(* Logix 5000 project; controller cal1632 1756-L62 rev 16.20; software revision 16.05; part 17 of 57 *)
(* tags used below, declared in another part *)
   AFI : BOOL;
   FAULT : BOOL;
   p01_param_fan_zero_speed : REAL;
   p01_param_open_oven_exh_sp : REAL;
   p01_param_open_oven_temp : REAL;
   p01_recipe_active : recipe;
   p01r02 : routine;
   p01r09_open_oven : BOOL;
   p01r09_pb_global_reset : BOOL;
   p01r13_permissive_oxidizer : BOOL;
   p02_dint_from_hmi : hmi_dint;
   p11r02_shutdown_temp : BOOL;
   p11r30 : routine;
   p11r30_request_heat : BOOL;
   p12_ai_exhaust_rpm : REAL;
   p12_ai_lfl : REAL;
   p12_ai_tc01 : REAL;
   p12_ai_tc02 : REAL;
   p12_ao_cv : REAL;
   p12_ao_exhaust_selected_speed : REAL;
   p12_di_burner_auto : BOOL;
   p12_di_burner_safeties_ok : BOOL;
   p12_di_door_open : BOOL;
   p12_di_exh : acs800_di_normal;
   p12_di_exh_fan_mtr_ts : BOOL;
   p12_di_exh_flow_ok : BOOL;
   p12_di_flame_failure : BOOL;
   p12_di_flame_on : BOOL;
   p12_di_fresh_air_clean : BOOL;
   p12_di_high_limit_temp_ok : BOOL;
   p12_di_recirc : acs800_di_normal;
   p12_di_recirc_flow_ok : BOOL;
   p12_di_sp0 : BOOL;
   p12_di_sp1 : BOOL;
   p12_di_tc01_bo : BOOL;
   p12_di_tc02_bo : BOOL;
   p12_di_zone_air_clean : BOOL;
   p12_do_enable_burner : BOOL;
   p12_do_exh : acs800_do_normal;
   p12_do_rst_flame : BOOL;
   p12_param_fast_to_soak : REAL;
   p12_param_lfl_hhl : REAL;
   p12_param_lfl_hl : REAL;
   p12_param_pid1_ff : REAL;
   p12_param_pid1_kd : REAL;
   p12_param_pid1_ki : REAL;
   p12_param_pid1_kp : REAL;
   p12_param_pid2_ff : REAL;
   p12_param_pid2_kd : REAL;
   p12_param_pid2_ki : REAL;
   p12_param_pid2_kp : REAL;
   p12_param_soak_to_fast : REAL;
   p12_param_tc01_dev : REAL;
   p12_param_tc01_hl : REAL;
   p12r02_shutdown_temp : BOOL;
   p12r16_pid_temp_cv : DINT;
   p12r16_temp_ok : BOOL;
   p12r20_safeties_ok : BOOL;
   p12r20_state : DINT;
   p12r30 : routine;
   p12r30_cv_man_sp : REAL;
   p12r30_pb_auto : BOOL;
   p12r30_pb_manual : BOOL;
   p12r30_pb_zone_off : BOOL;
   p12r30_pb_zone_on : BOOL;
   p12r30_permissive_run : BOOL;
   p12r30_pid_temp : PID;
   p12r30_pid_temp_pv : REAL;
   p12r30_pid_temp_sp : REAL;
   p12r30_pid_temp_sp_error : REAL;
   p12r30_pid_temp_sp_last : REAL;
   p12r30_request_deviation_warning : BOOL;
   p12r30_request_heat : BOOL;
   p12r30_request_heat_last : BOOL;
   p12r30_request_manual : BOOL;
   p12r30_request_PID_shot : BOOL;
   p12r30_request_soak_control : BOOL;
   p12r30_temp_deviation_setpoint : DINT;
   p12r30_timer_fault : TIMER[16];
   p12r30_timer_warning : TIMER[12];
   p12r30_vfds_ok : BOOL;
   p12r31 : routine;
   p12r31_pb_start : BOOL;
   p12r31_pb_stop : BOOL;
   p12r31_request_auto_run : BOOL;
   p12r31_run_permissive : BOOL;
   p12r31_timer_fault : TIMER[5];
   p12r31_timer_warning : TIMER[5];
   p12r31_vfd_stopped : BOOL;
   p12r32 : routine;
   p23_di_exhaust_speed_ok : BOOL;
   p23_di_impreg_exhaust_running : BOOL;
   p23_di_impreg_tank_up : BOOL;
   p23_di_supply_speed_ok : BOOL;
   p23r02 : routine;
   p23r13 : routine;
(* P12_Zone_2, continued *)

ROUTINE R30_Temperature_Control   (* ladder *)
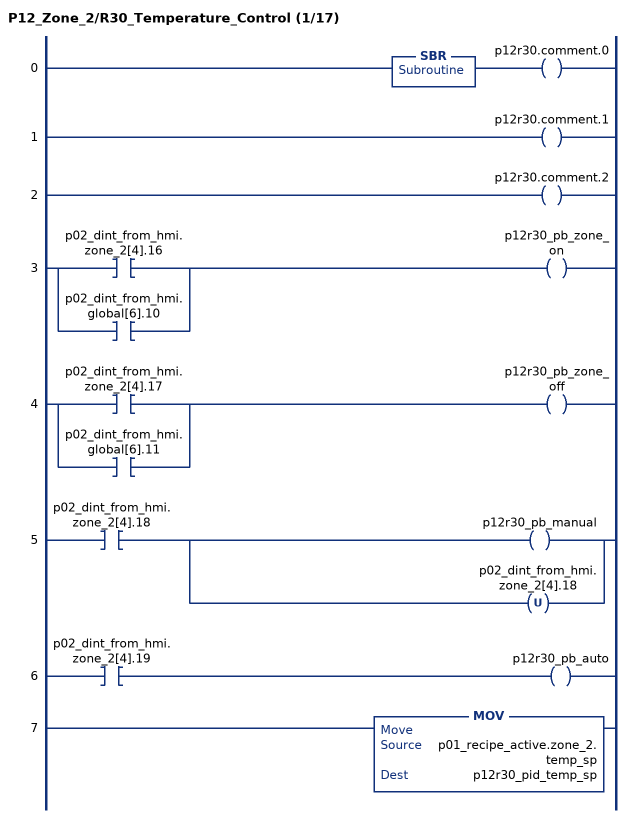
   0: SBR()OTE(p12r30.comment.0);
   1: OTE(p12r30.comment.1);
   2: OTE(p12r30.comment.2);
   3: [XIC(p02_dint_from_hmi.zone_2[4].16) ,XIC(p02_dint_from_hmi.global[6].10) ]OTE(p12r30_pb_zone_on);
   4: [XIC(p02_dint_from_hmi.zone_2[4].17) ,XIC(p02_dint_from_hmi.global[6].11) ]OTE(p12r30_pb_zone_off);
   5: XIC(p02_dint_from_hmi.zone_2[4].18)[OTE(p12r30_pb_manual) ,OTU(p02_dint_from_hmi.zone_2[4].18) ];
   6: XIC(p02_dint_from_hmi.zone_2[4].19)OTE(p12r30_pb_auto);
   7: MOV(p01_recipe_active.zone_2.temp_sp,p12r30_pid_temp_sp);
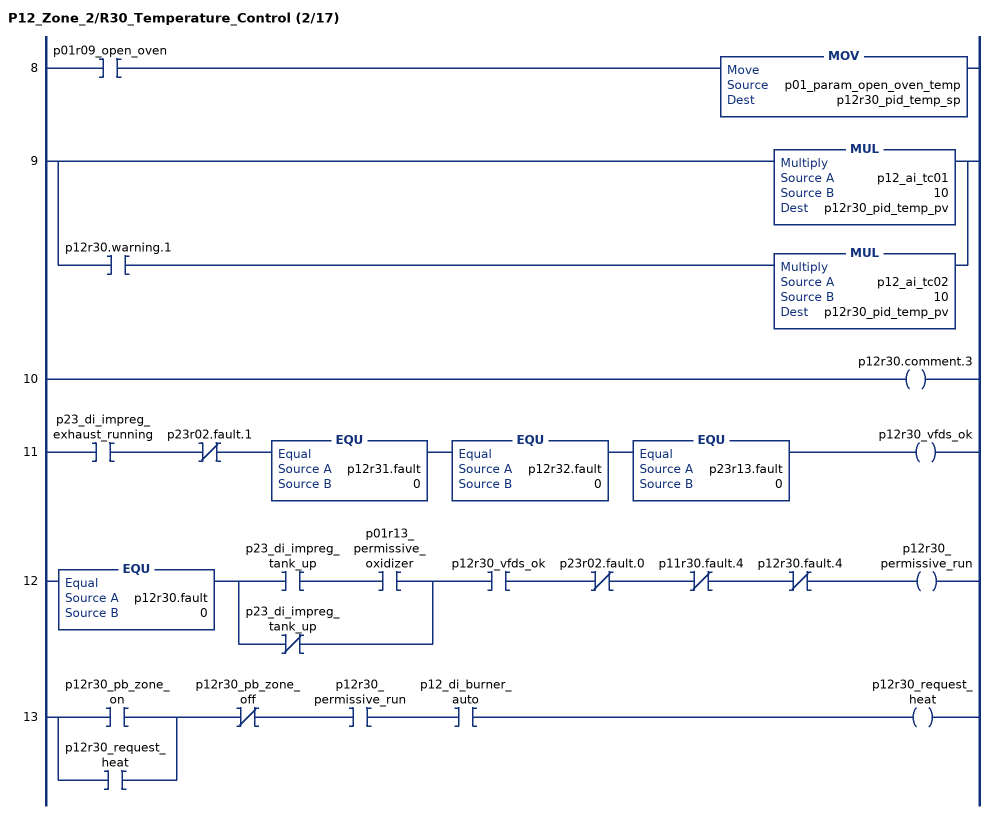
   8: XIC(p01r09_open_oven)MOV(p01_param_open_oven_temp,p12r30_pid_temp_sp);
   9: [MUL(p12_ai_tc01,10,p12r30_pid_temp_pv) ,XIC(p12r30.warning.1) MUL(p12_ai_tc02,10,p12r30_pid_temp_pv) ];
   10: OTE(p12r30.comment.3);
   11: XIC(p23_di_impreg_exhaust_running)XIO(p23r02.fault.1)EQU(p12r31.fault,0)EQU(p12r32.fault,0)EQU(p23r13.fault,0)OTE(p12r30_vfds_ok);
   12: EQU(p12r30.fault,0)[XIC(p23_di_impreg_tank_up) XIC(p01r13_permissive_oxidizer) ,XIO(p23_di_impreg_tank_up) ]XIC(p12r30_vfds_ok)XIO(p23r02.fault.0)XIO(p11r30.fault.4)XIO(p12r30.fault.4)OTE(p12r30_permissive_run);
   13: [XIC(p12r30_pb_zone_on) ,XIC(p12r30_request_heat) ]XIO(p12r30_pb_zone_off)XIC(p12r30_permissive_run)XIC(p12_di_burner_auto)OTE(p12r30_request_heat);
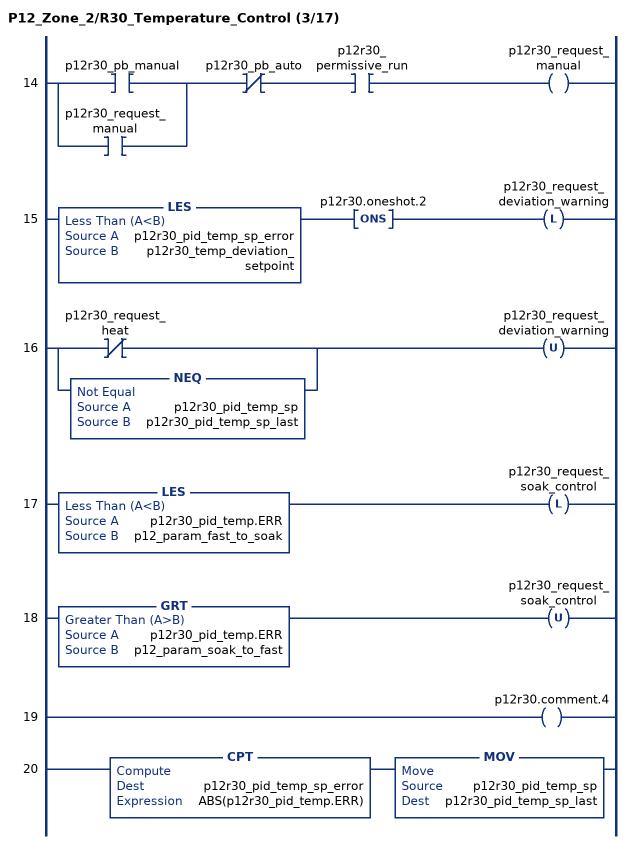
   14: [XIC(p12r30_pb_manual) ,XIC(p12r30_request_manual) ]XIO(p12r30_pb_auto)XIC(p12r30_permissive_run)OTE(p12r30_request_manual);
   15: LES(p12r30_pid_temp_sp_error,p12r30_temp_deviation_setpoint)ONS(p12r30.oneshot.2)OTL(p12r30_request_deviation_warning);
   16: [XIO(p12r30_request_heat) ,NEQ(p12r30_pid_temp_sp,p12r30_pid_temp_sp_last) ]OTU(p12r30_request_deviation_warning);
   17: LES(p12r30_pid_temp.ERR,p12_param_fast_to_soak)OTL(p12r30_request_soak_control);
   18: GRT(p12r30_pid_temp.ERR,p12_param_soak_to_fast)OTU(p12r30_request_soak_control);
   19: OTE(p12r30.comment.4);
   20: CPT(p12r30_pid_temp_sp_error,ABS(p12r30_pid_temp.ERR))MOV(p12r30_pid_temp_sp,p12r30_pid_temp_sp_last);
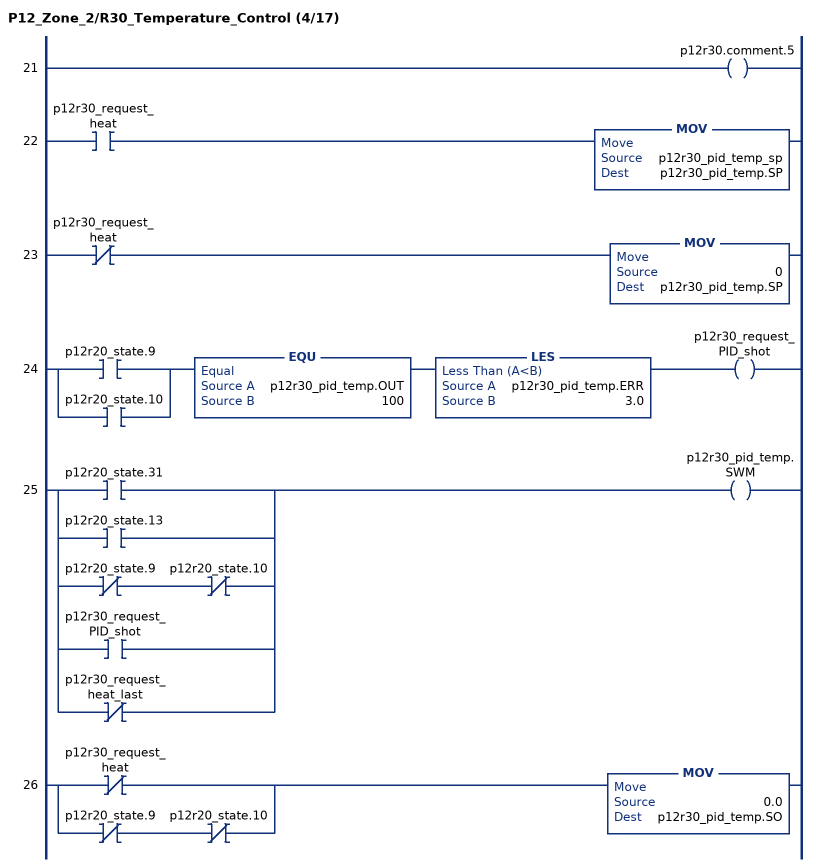
   21: OTE(p12r30.comment.5);
   22: XIC(p12r30_request_heat)MOV(p12r30_pid_temp_sp,p12r30_pid_temp.SP);
   23: XIO(p12r30_request_heat)MOV(0,p12r30_pid_temp.SP);
   24: [XIC(p12r20_state.9) ,XIC(p12r20_state.10) ]EQU(p12r30_pid_temp.OUT,100)LES(p12r30_pid_temp.ERR,3.0)OTE(p12r30_request_PID_shot);
   25: [XIC(p12r20_state.31) ,XIC(p12r20_state.13) ,XIO(p12r20_state.9) XIO(p12r20_state.10) ,XIC(p12r30_request_PID_shot) ,XIO(p12r30_request_heat_last) ]OTE(p12r30_pid_temp.SWM);
   26: [XIO(p12r30_request_heat) ,XIO(p12r20_state.9) XIO(p12r20_state.10) ]MOV(0.0,p12r30_pid_temp.SO);
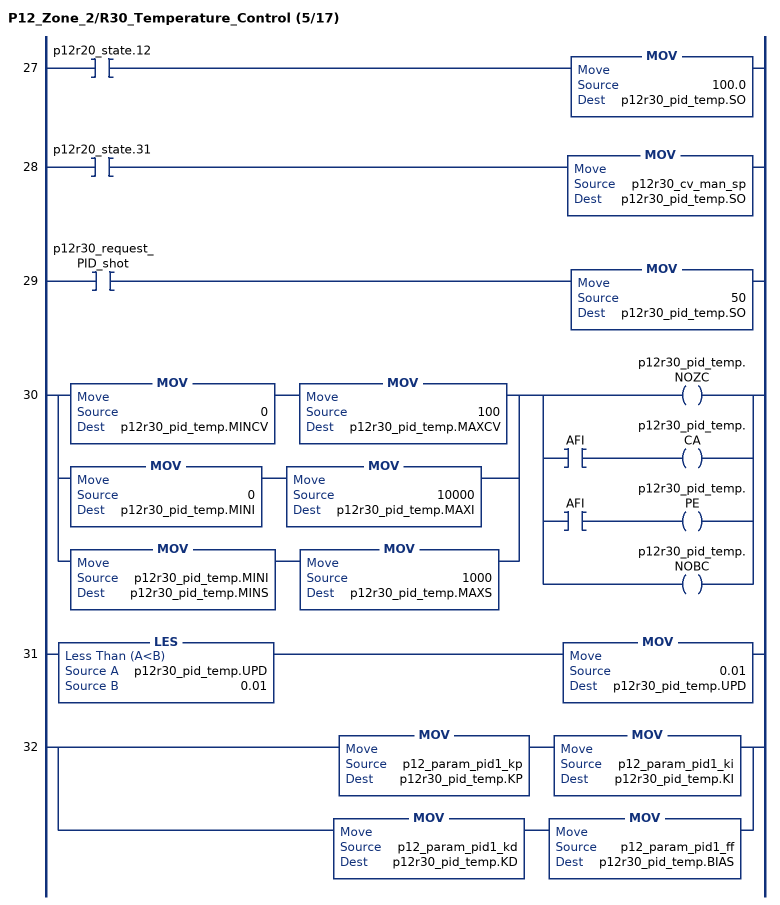
   27: XIC(p12r20_state.12)MOV(100.0,p12r30_pid_temp.SO);
   28: XIC(p12r20_state.31)MOV(p12r30_cv_man_sp,p12r30_pid_temp.SO);
   29: XIC(p12r30_request_PID_shot)MOV(50,p12r30_pid_temp.SO);
   30: [MOV(0,p12r30_pid_temp.MINCV) MOV(100,p12r30_pid_temp.MAXCV) ,MOV(0,p12r30_pid_temp.MINI) MOV(10000,p12r30_pid_temp.MAXI) ,MOV(p12r30_pid_temp.MINI,p12r30_pid_temp.MINS) MOV(1000,p12r30_pid_temp.MAXS) ][OTE(p12r30_pid_temp.NOZC) ,XIC(AFI) OTE(p12r30_pid_temp.CA) ,XIC(AFI) OTE(p12r30_pid_temp.PE) ,OTE(p12r30_pid_temp.NOBC) ];
   31: LES(p12r30_pid_temp.UPD,0.01)MOV(0.01,p12r30_pid_temp.UPD);
   32: [MOV(p12_param_pid1_kp,p12r30_pid_temp.KP) MOV(p12_param_pid1_ki,p12r30_pid_temp.KI) ,MOV(p12_param_pid1_kd,p12r30_pid_temp.KD) MOV(p12_param_pid1_ff,p12r30_pid_temp.BIAS) ];
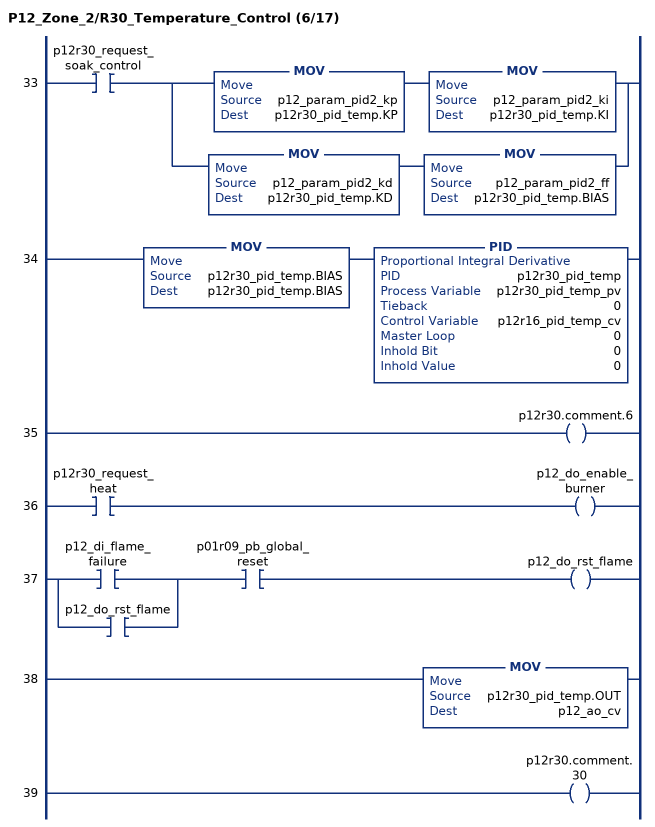
   33: XIC(p12r30_request_soak_control)[MOV(p12_param_pid2_kp,p12r30_pid_temp.KP) MOV(p12_param_pid2_ki,p12r30_pid_temp.KI) ,MOV(p12_param_pid2_kd,p12r30_pid_temp.KD) MOV(p12_param_pid2_ff,p12r30_pid_temp.BIAS) ];
   34: MOV(p12r30_pid_temp.BIAS,p12r30_pid_temp.BIAS)PID(p12r30_pid_temp,p12r30_pid_temp_pv,0,p12r16_pid_temp_cv,0,0,0);
   35: OTE(p12r30.comment.6);
   36: XIC(p12r30_request_heat)OTE(p12_do_enable_burner);
   37: [XIC(p12_di_flame_failure) ,XIC(p12_do_rst_flame) ]XIC(p01r09_pb_global_reset)OTE(p12_do_rst_flame);
   38: MOV(p12r30_pid_temp.OUT,p12_ao_cv);
   39: OTE(p12r30.comment.30);
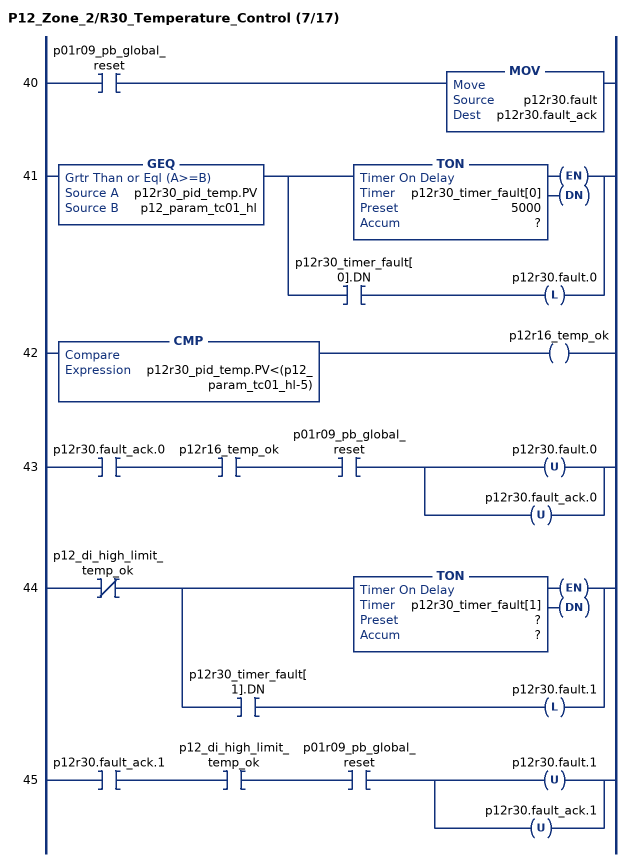
   40: XIC(p01r09_pb_global_reset)MOV(p12r30.fault,p12r30.fault_ack);
   41: GEQ(p12r30_pid_temp.PV,p12_param_tc01_hl)[TON(p12r30_timer_fault[0],?,?) ,XIC(p12r30_timer_fault[0].DN) OTL(p12r30.fault.0) ];
   42: CMP(p12r30_pid_temp.PV<(p12_param_tc01_hl-5))OTE(p12r16_temp_ok);
   43: XIC(p12r30.fault_ack.0)XIC(p12r16_temp_ok)XIC(p01r09_pb_global_reset)[OTU(p12r30.fault.0) ,OTU(p12r30.fault_ack.0) ];
   44: XIO(p12_di_high_limit_temp_ok)[TON(p12r30_timer_fault[1],?,?) ,XIC(p12r30_timer_fault[1].DN) OTL(p12r30.fault.1) ];
   45: XIC(p12r30.fault_ack.1)XIC(p12_di_high_limit_temp_ok)XIC(p01r09_pb_global_reset)[OTU(p12r30.fault.1) ,OTU(p12r30.fault_ack.1) ];
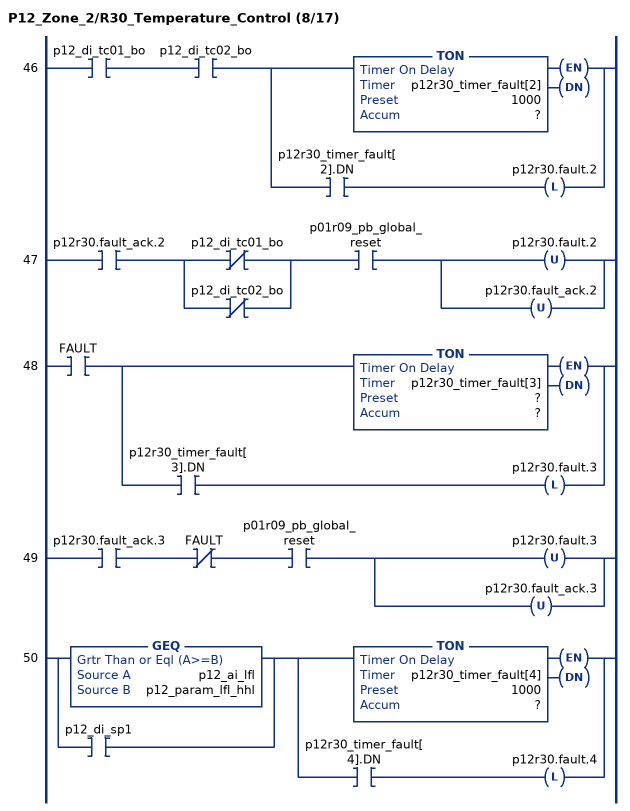
   46: XIC(p12_di_tc01_bo)XIC(p12_di_tc02_bo)[TON(p12r30_timer_fault[2],?,?) ,XIC(p12r30_timer_fault[2].DN) OTL(p12r30.fault.2) ];
   47: XIC(p12r30.fault_ack.2)[XIO(p12_di_tc01_bo) ,XIO(p12_di_tc02_bo) ]XIC(p01r09_pb_global_reset)[OTU(p12r30.fault.2) ,OTU(p12r30.fault_ack.2) ];
   48: XIC(FAULT)[TON(p12r30_timer_fault[3],?,?) ,XIC(p12r30_timer_fault[3].DN) OTL(p12r30.fault.3) ];
   49: XIC(p12r30.fault_ack.3)XIO(FAULT)XIC(p01r09_pb_global_reset)[OTU(p12r30.fault.3) ,OTU(p12r30.fault_ack.3) ];
   50: [GEQ(p12_ai_lfl,p12_param_lfl_hhl) ,XIC(p12_di_sp1) ][TON(p12r30_timer_fault[4],?,?) ,XIC(p12r30_timer_fault[4].DN) OTL(p12r30.fault.4) ];
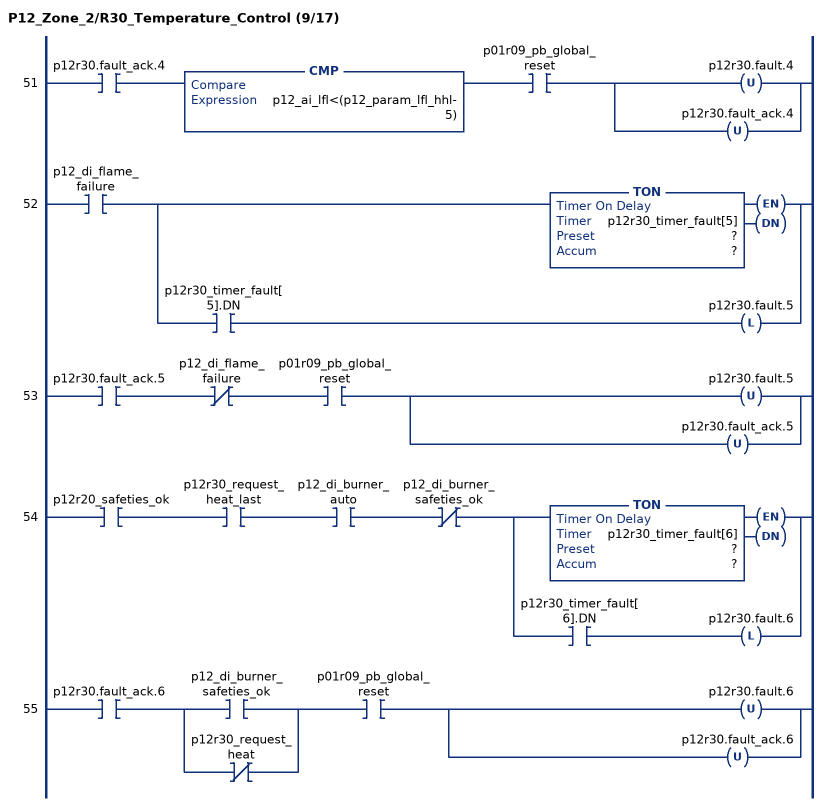
   51: XIC(p12r30.fault_ack.4)CMP(p12_ai_lfl<(p12_param_lfl_hhl-5))XIC(p01r09_pb_global_reset)[OTU(p12r30.fault.4) ,OTU(p12r30.fault_ack.4) ];
   52: XIC(p12_di_flame_failure)[TON(p12r30_timer_fault[5],?,?) ,XIC(p12r30_timer_fault[5].DN) OTL(p12r30.fault.5) ];
   53: XIC(p12r30.fault_ack.5)XIO(p12_di_flame_failure)XIC(p01r09_pb_global_reset)[OTU(p12r30.fault.5) ,OTU(p12r30.fault_ack.5) ];
   54: XIC(p12r20_safeties_ok)XIC(p12r30_request_heat_last)XIC(p12_di_burner_auto)XIO(p12_di_burner_safeties_ok)[TON(p12r30_timer_fault[6],?,?) ,XIC(p12r30_timer_fault[6].DN) OTL(p12r30.fault.6) ];
   55: XIC(p12r30.fault_ack.6)[XIC(p12_di_burner_safeties_ok) ,XIO(p12r30_request_heat) ]XIC(p01r09_pb_global_reset)[OTU(p12r30.fault.6) ,OTU(p12r30.fault_ack.6) ];
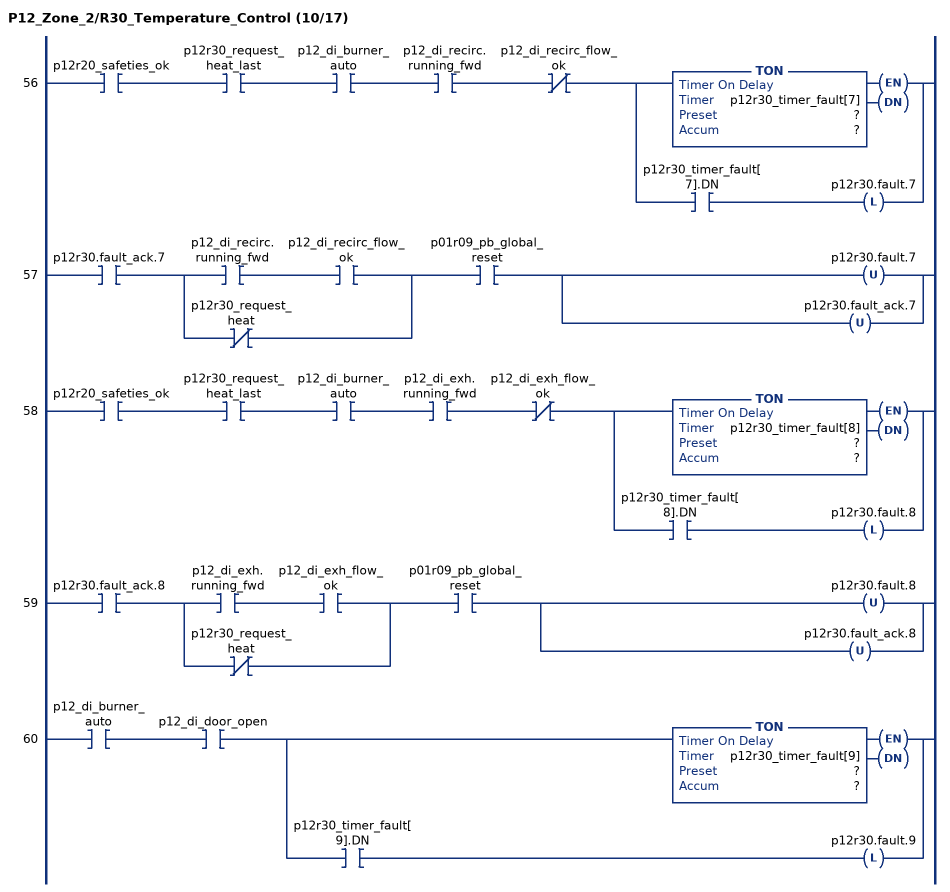
   56: XIC(p12r20_safeties_ok)XIC(p12r30_request_heat_last)XIC(p12_di_burner_auto)XIC(p12_di_recirc.running_fwd)XIO(p12_di_recirc_flow_ok)[TON(p12r30_timer_fault[7],?,?) ,XIC(p12r30_timer_fault[7].DN) OTL(p12r30.fault.7) ];
   57: XIC(p12r30.fault_ack.7)[XIC(p12_di_recirc.running_fwd) XIC(p12_di_recirc_flow_ok) ,XIO(p12r30_request_heat) ]XIC(p01r09_pb_global_reset)[OTU(p12r30.fault.7) ,OTU(p12r30.fault_ack.7) ];
   58: XIC(p12r20_safeties_ok)XIC(p12r30_request_heat_last)XIC(p12_di_burner_auto)XIC(p12_di_exh.running_fwd)XIO(p12_di_exh_flow_ok)[TON(p12r30_timer_fault[8],?,?) ,XIC(p12r30_timer_fault[8].DN) OTL(p12r30.fault.8) ];
   59: XIC(p12r30.fault_ack.8)[XIC(p12_di_exh.running_fwd) XIC(p12_di_exh_flow_ok) ,XIO(p12r30_request_heat) ]XIC(p01r09_pb_global_reset)[OTU(p12r30.fault.8) ,OTU(p12r30.fault_ack.8) ];
   60: XIC(p12_di_burner_auto)XIC(p12_di_door_open)[TON(p12r30_timer_fault[9],?,?) ,XIC(p12r30_timer_fault[9].DN) OTL(p12r30.fault.9) ];
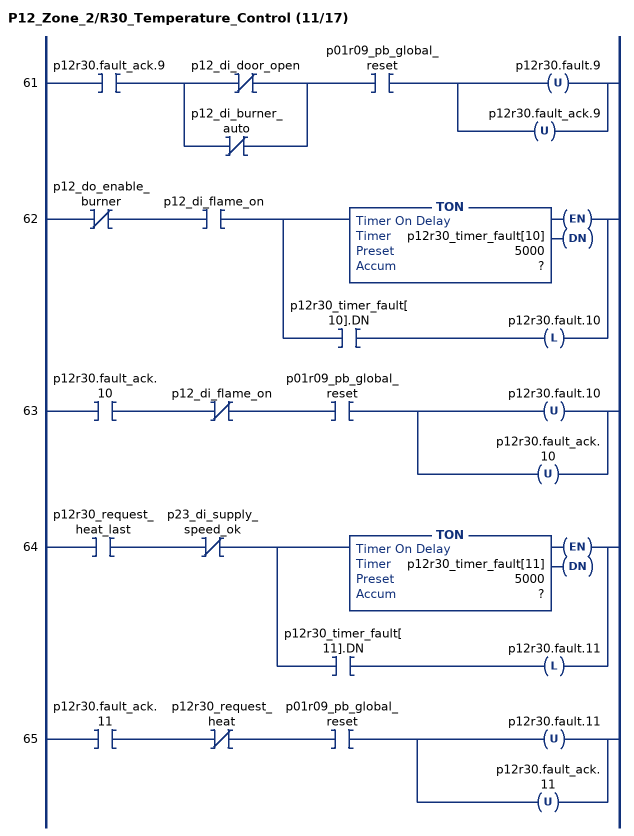
   61: XIC(p12r30.fault_ack.9)[XIO(p12_di_door_open) ,XIO(p12_di_burner_auto) ]XIC(p01r09_pb_global_reset)[OTU(p12r30.fault.9) ,OTU(p12r30.fault_ack.9) ];
   62: XIO(p12_do_enable_burner)XIC(p12_di_flame_on)[TON(p12r30_timer_fault[10],?,?) ,XIC(p12r30_timer_fault[10].DN) OTL(p12r30.fault.10) ];
   63: XIC(p12r30.fault_ack.10)XIO(p12_di_flame_on)XIC(p01r09_pb_global_reset)[OTU(p12r30.fault.10) ,OTU(p12r30.fault_ack.10) ];
   64: XIC(p12r30_request_heat_last)XIO(p23_di_supply_speed_ok)[TON(p12r30_timer_fault[11],?,?) ,XIC(p12r30_timer_fault[11].DN) OTL(p12r30.fault.11) ];
   65: XIC(p12r30.fault_ack.11)XIO(p12r30_request_heat)XIC(p01r09_pb_global_reset)[OTU(p12r30.fault.11) ,OTU(p12r30.fault_ack.11) ];
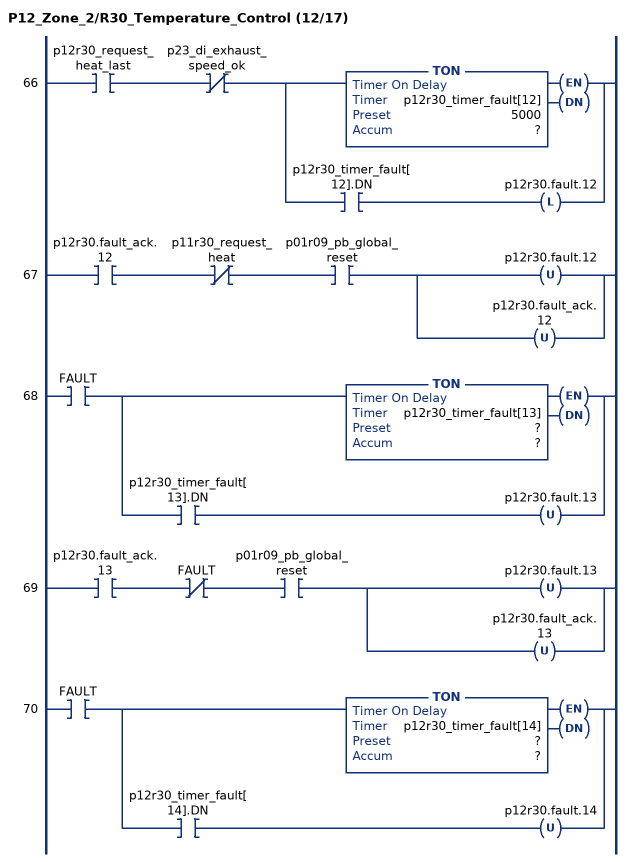
   66: XIC(p12r30_request_heat_last)XIO(p23_di_exhaust_speed_ok)[TON(p12r30_timer_fault[12],?,?) ,XIC(p12r30_timer_fault[12].DN) OTL(p12r30.fault.12) ];
   67: XIC(p12r30.fault_ack.12)XIO(p11r30_request_heat)XIC(p01r09_pb_global_reset)[OTU(p12r30.fault.12) ,OTU(p12r30.fault_ack.12) ];
   68: XIC(FAULT)[TON(p12r30_timer_fault[13],?,?) ,XIC(p12r30_timer_fault[13].DN) OTU(p12r30.fault.13) ];
   69: XIC(p12r30.fault_ack.13)XIO(FAULT)XIC(p01r09_pb_global_reset)[OTU(p12r30.fault.13) ,OTU(p12r30.fault_ack.13) ];
   70: XIC(FAULT)[TON(p12r30_timer_fault[14],?,?) ,XIC(p12r30_timer_fault[14].DN) OTU(p12r30.fault.14) ];
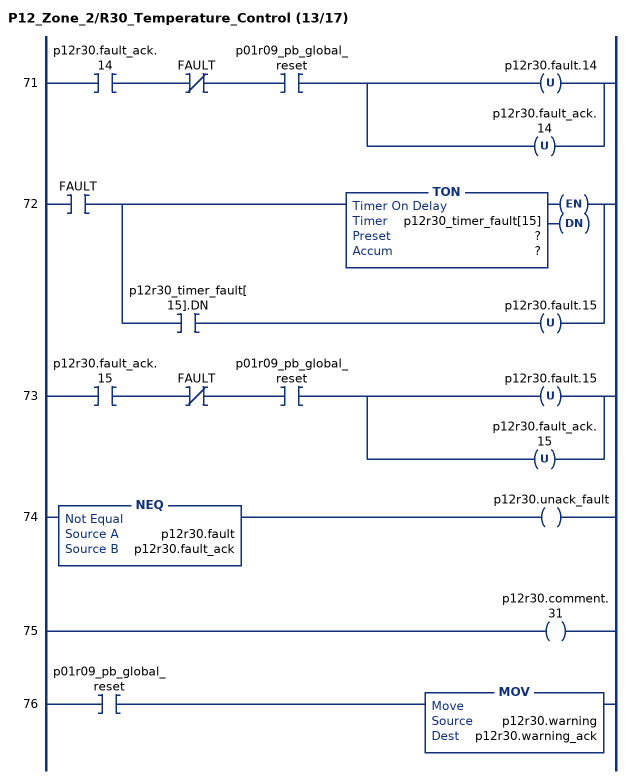
   71: XIC(p12r30.fault_ack.14)XIO(FAULT)XIC(p01r09_pb_global_reset)[OTU(p12r30.fault.14) ,OTU(p12r30.fault_ack.14) ];
   72: XIC(FAULT)[TON(p12r30_timer_fault[15],?,?) ,XIC(p12r30_timer_fault[15].DN) OTU(p12r30.fault.15) ];
   73: XIC(p12r30.fault_ack.15)XIO(FAULT)XIC(p01r09_pb_global_reset)[OTU(p12r30.fault.15) ,OTU(p12r30.fault_ack.15) ];
   74: NEQ(p12r30.fault,p12r30.fault_ack)OTE(p12r30.unack_fault);
   75: OTE(p12r30.comment.31);
   76: XIC(p01r09_pb_global_reset)MOV(p12r30.warning,p12r30.warning_ack);
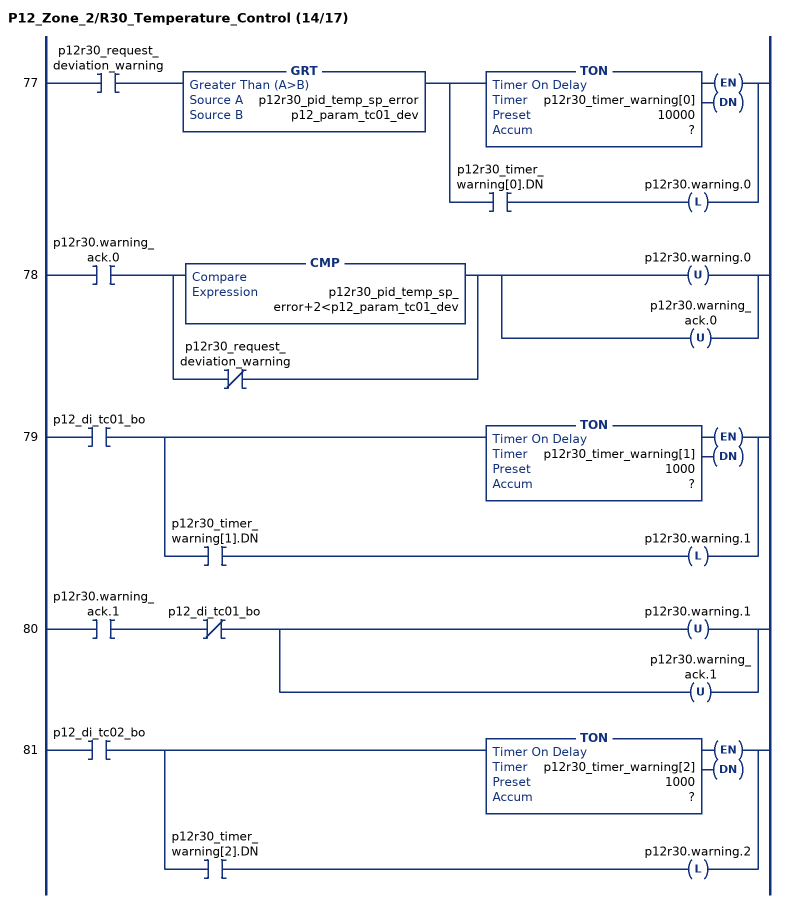
   77: XIC(p12r30_request_deviation_warning)GRT(p12r30_pid_temp_sp_error,p12_param_tc01_dev)[TON(p12r30_timer_warning[0],?,?) ,XIC(p12r30_timer_warning[0].DN) OTL(p12r30.warning.0) ];
   78: XIC(p12r30.warning_ack.0)[CMP(p12r30_pid_temp_sp_error+2<p12_param_tc01_dev) ,XIO(p12r30_request_deviation_warning) ][OTU(p12r30.warning.0) ,OTU(p12r30.warning_ack.0) ];
   79: XIC(p12_di_tc01_bo)[TON(p12r30_timer_warning[1],?,?) ,XIC(p12r30_timer_warning[1].DN) OTL(p12r30.warning.1) ];
   80: XIC(p12r30.warning_ack.1)XIO(p12_di_tc01_bo)[OTU(p12r30.warning.1) ,OTU(p12r30.warning_ack.1) ];
   81: XIC(p12_di_tc02_bo)[TON(p12r30_timer_warning[2],?,?) ,XIC(p12r30_timer_warning[2].DN) OTL(p12r30.warning.2) ];
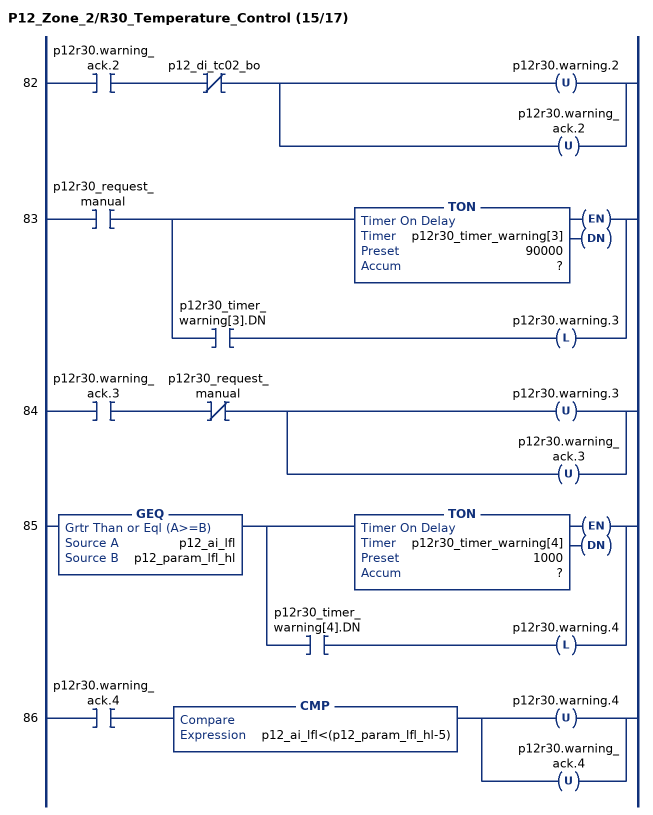
   82: XIC(p12r30.warning_ack.2)XIO(p12_di_tc02_bo)[OTU(p12r30.warning.2) ,OTU(p12r30.warning_ack.2) ];
   83: XIC(p12r30_request_manual)[TON(p12r30_timer_warning[3],?,?) ,XIC(p12r30_timer_warning[3].DN) OTL(p12r30.warning.3) ];
   84: XIC(p12r30.warning_ack.3)XIO(p12r30_request_manual)[OTU(p12r30.warning.3) ,OTU(p12r30.warning_ack.3) ];
   85: GEQ(p12_ai_lfl,p12_param_lfl_hl)[TON(p12r30_timer_warning[4],?,?) ,XIC(p12r30_timer_warning[4].DN) OTL(p12r30.warning.4) ];
   86: XIC(p12r30.warning_ack.4)CMP(p12_ai_lfl<(p12_param_lfl_hl-5))[OTU(p12r30.warning.4) ,OTU(p12r30.warning_ack.4) ];
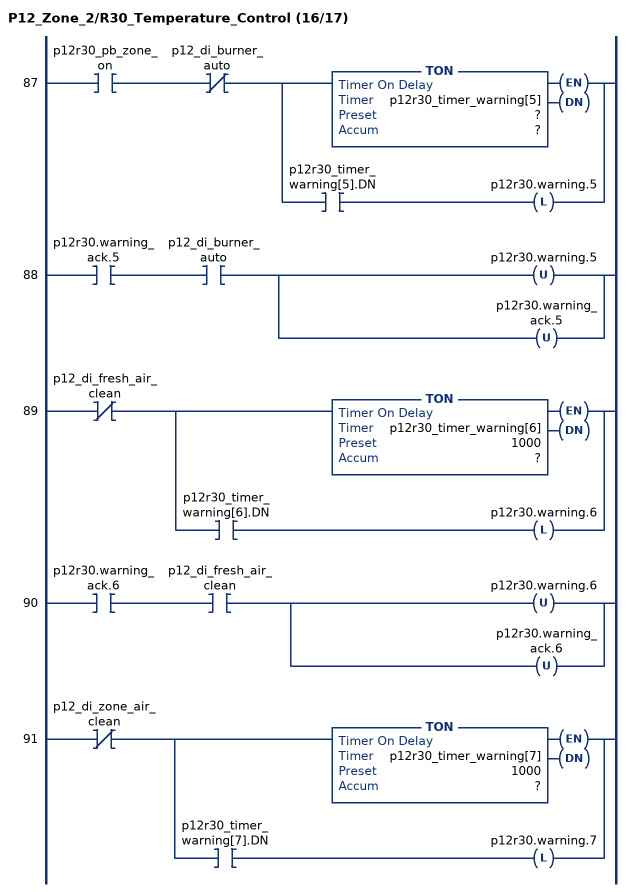
   87: XIC(p12r30_pb_zone_on)XIO(p12_di_burner_auto)[TON(p12r30_timer_warning[5],?,?) ,XIC(p12r30_timer_warning[5].DN) OTL(p12r30.warning.5) ];
   88: XIC(p12r30.warning_ack.5)XIC(p12_di_burner_auto)[OTU(p12r30.warning.5) ,OTU(p12r30.warning_ack.5) ];
   89: XIO(p12_di_fresh_air_clean)[TON(p12r30_timer_warning[6],?,?) ,XIC(p12r30_timer_warning[6].DN) OTL(p12r30.warning.6) ];
   90: XIC(p12r30.warning_ack.6)XIC(p12_di_fresh_air_clean)[OTU(p12r30.warning.6) ,OTU(p12r30.warning_ack.6) ];
   91: XIO(p12_di_zone_air_clean)[TON(p12r30_timer_warning[7],?,?) ,XIC(p12r30_timer_warning[7].DN) OTL(p12r30.warning.7) ];
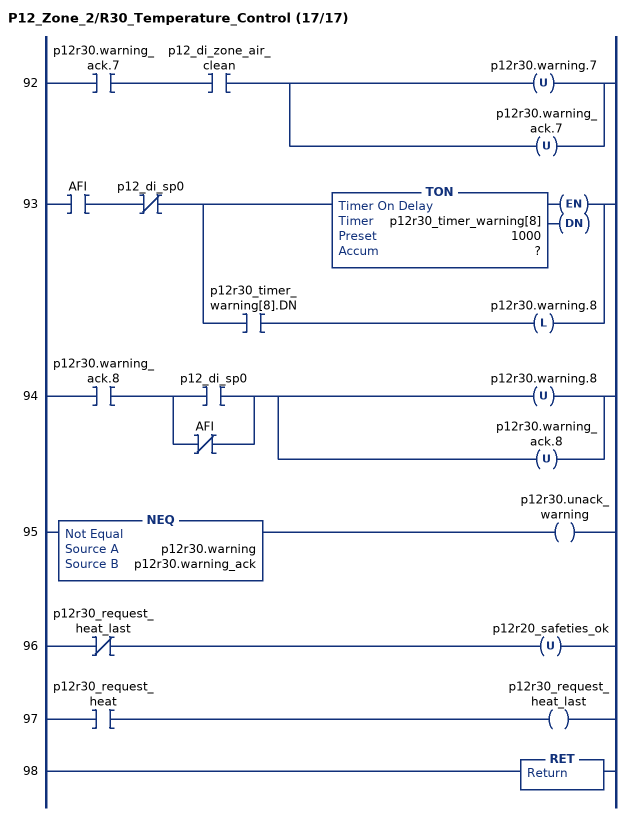
   92: XIC(p12r30.warning_ack.7)XIC(p12_di_zone_air_clean)[OTU(p12r30.warning.7) ,OTU(p12r30.warning_ack.7) ];
   93: XIC(AFI)XIO(p12_di_sp0)[TON(p12r30_timer_warning[8],?,?) ,XIC(p12r30_timer_warning[8].DN) OTL(p12r30.warning.8) ];
   94: XIC(p12r30.warning_ack.8)[XIC(p12_di_sp0) ,XIO(AFI) ][OTU(p12r30.warning.8) ,OTU(p12r30.warning_ack.8) ];
   95: NEQ(p12r30.warning,p12r30.warning_ack)OTE(p12r30.unack_warning);
   96: XIO(p12r30_request_heat_last)OTU(p12r20_safeties_ok);
   97: XIC(p12r30_request_heat)OTE(p12r30_request_heat_last);
   98: RET();
END_ROUTINE

ROUTINE R31_Exhaust_VFD   (* ladder *)
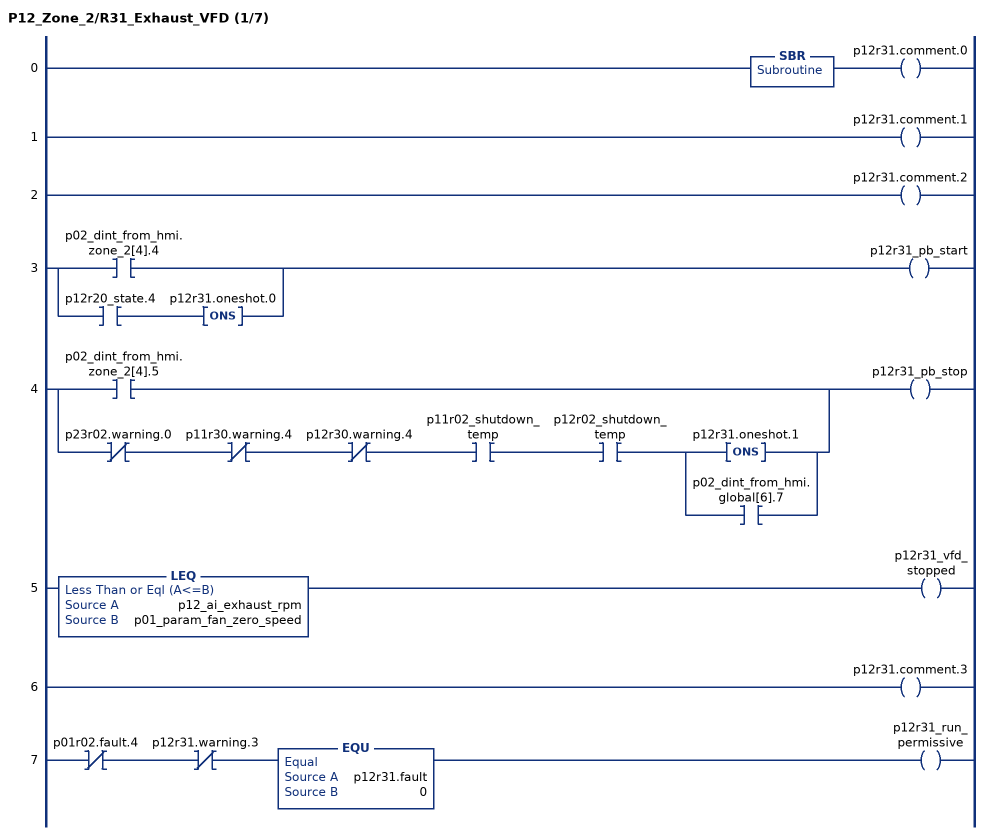
   0: SBR()OTE(p12r31.comment.0);
   1: OTE(p12r31.comment.1);
   2: OTE(p12r31.comment.2);
   3: [XIC(p02_dint_from_hmi.zone_2[4].4) ,XIC(p12r20_state.4) ONS(p12r31.oneshot.0) ]OTE(p12r31_pb_start);
   4: [XIC(p02_dint_from_hmi.zone_2[4].5) ,XIO(p23r02.warning.0) XIO(p11r30.warning.4) XIO(p12r30.warning.4) XIC(p11r02_shutdown_temp) XIC(p12r02_shutdown_temp) [ONS(p12r31.oneshot.1) ,XIC(p02_dint_from_hmi.global[6].7) ] ]OTE(p12r31_pb_stop);
   5: LEQ(p12_ai_exhaust_rpm,p01_param_fan_zero_speed)OTE(p12r31_vfd_stopped);
   6: OTE(p12r31.comment.3);
   7: XIO(p01r02.fault.4)XIO(p12r31.warning.3)EQU(p12r31.fault,0)OTE(p12r31_run_permissive);
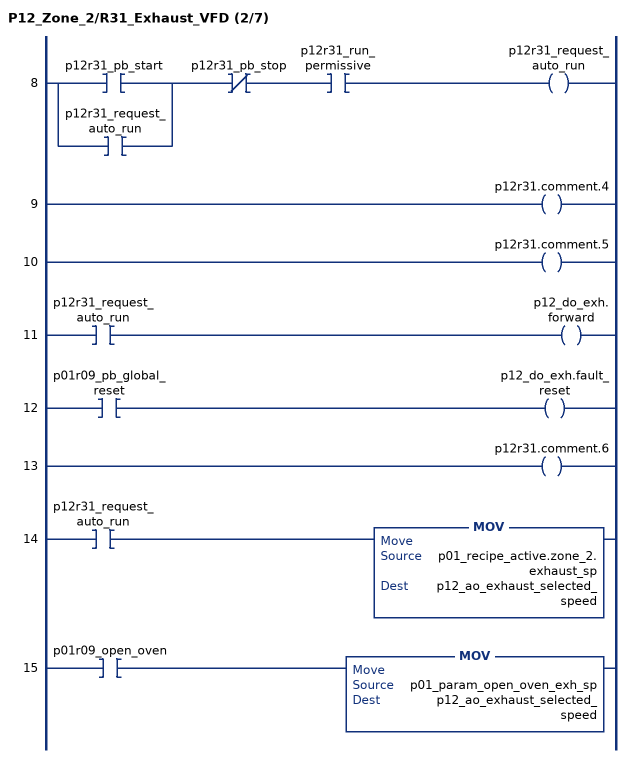
   8: [XIC(p12r31_pb_start) ,XIC(p12r31_request_auto_run) ]XIO(p12r31_pb_stop)XIC(p12r31_run_permissive)OTE(p12r31_request_auto_run);
   9: OTE(p12r31.comment.4);
   10: OTE(p12r31.comment.5);
   11: XIC(p12r31_request_auto_run)OTE(p12_do_exh.forward);
   12: XIC(p01r09_pb_global_reset)OTE(p12_do_exh.fault_reset);
   13: OTE(p12r31.comment.6);
   14: XIC(p12r31_request_auto_run)MOV(p01_recipe_active.zone_2.exhaust_sp,p12_ao_exhaust_selected_speed);
   15: XIC(p01r09_open_oven)MOV(p01_param_open_oven_exh_sp,p12_ao_exhaust_selected_speed);
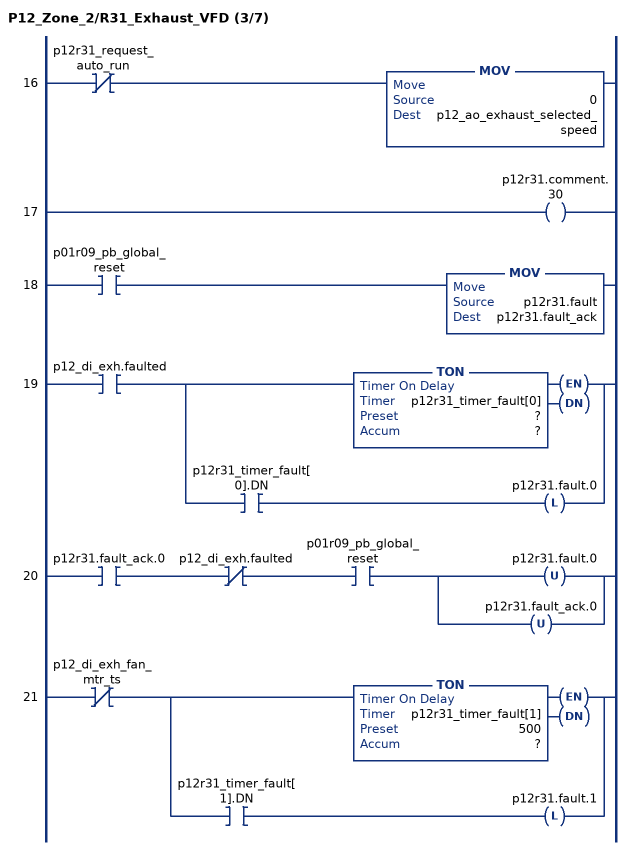
   16: XIO(p12r31_request_auto_run)MOV(0,p12_ao_exhaust_selected_speed);
   17: OTE(p12r31.comment.30);
   18: XIC(p01r09_pb_global_reset)MOV(p12r31.fault,p12r31.fault_ack);
   19: XIC(p12_di_exh.faulted)[TON(p12r31_timer_fault[0],?,?) ,XIC(p12r31_timer_fault[0].DN) OTL(p12r31.fault.0) ];
   20: XIC(p12r31.fault_ack.0)XIO(p12_di_exh.faulted)XIC(p01r09_pb_global_reset)[OTU(p12r31.fault.0) ,OTU(p12r31.fault_ack.0) ];
   21: XIO(p12_di_exh_fan_mtr_ts)[TON(p12r31_timer_fault[1],?,?) ,XIC(p12r31_timer_fault[1].DN) OTL(p12r31.fault.1) ];
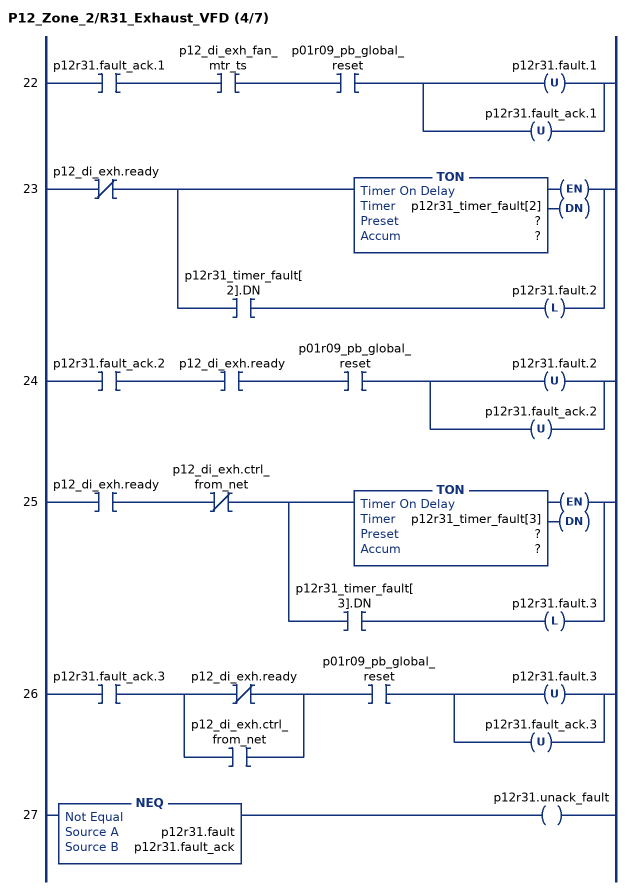
   22: XIC(p12r31.fault_ack.1)XIC(p12_di_exh_fan_mtr_ts)XIC(p01r09_pb_global_reset)[OTU(p12r31.fault.1) ,OTU(p12r31.fault_ack.1) ];
   23: XIO(p12_di_exh.ready)[TON(p12r31_timer_fault[2],?,?) ,XIC(p12r31_timer_fault[2].DN) OTL(p12r31.fault.2) ];
   24: XIC(p12r31.fault_ack.2)XIC(p12_di_exh.ready)XIC(p01r09_pb_global_reset)[OTU(p12r31.fault.2) ,OTU(p12r31.fault_ack.2) ];
   25: XIC(p12_di_exh.ready)XIO(p12_di_exh.ctrl_from_net)[TON(p12r31_timer_fault[3],?,?) ,XIC(p12r31_timer_fault[3].DN) OTL(p12r31.fault.3) ];
   26: XIC(p12r31.fault_ack.3)[XIO(p12_di_exh.ready) ,XIC(p12_di_exh.ctrl_from_net) ]XIC(p01r09_pb_global_reset)[OTU(p12r31.fault.3) ,OTU(p12r31.fault_ack.3) ];
   27: NEQ(p12r31.fault,p12r31.fault_ack)OTE(p12r31.unack_fault);
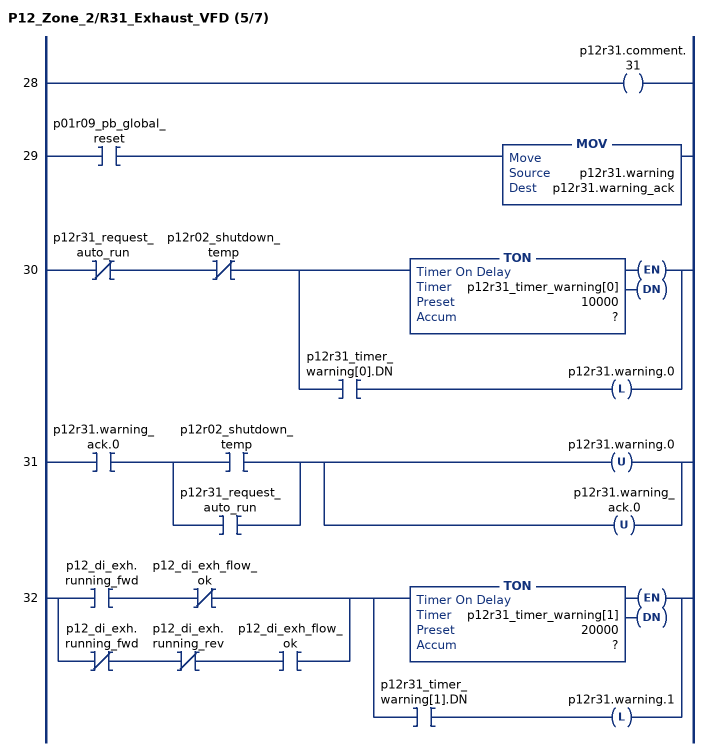
   28: OTE(p12r31.comment.31);
   29: XIC(p01r09_pb_global_reset)MOV(p12r31.warning,p12r31.warning_ack);
   30: XIO(p12r31_request_auto_run)XIO(p12r02_shutdown_temp)[TON(p12r31_timer_warning[0],?,?) ,XIC(p12r31_timer_warning[0].DN) OTL(p12r31.warning.0) ];
   31: XIC(p12r31.warning_ack.0)[XIC(p12r02_shutdown_temp) ,XIC(p12r31_request_auto_run) ][OTU(p12r31.warning.0) ,OTU(p12r31.warning_ack.0) ];
   32: [XIC(p12_di_exh.running_fwd) XIO(p12_di_exh_flow_ok) ,XIO(p12_di_exh.running_fwd) XIO(p12_di_exh.running_rev) XIC(p12_di_exh_flow_ok) ][TON(p12r31_timer_warning[1],?,?) ,XIC(p12r31_timer_warning[1].DN) OTL(p12r31.warning.1) ];
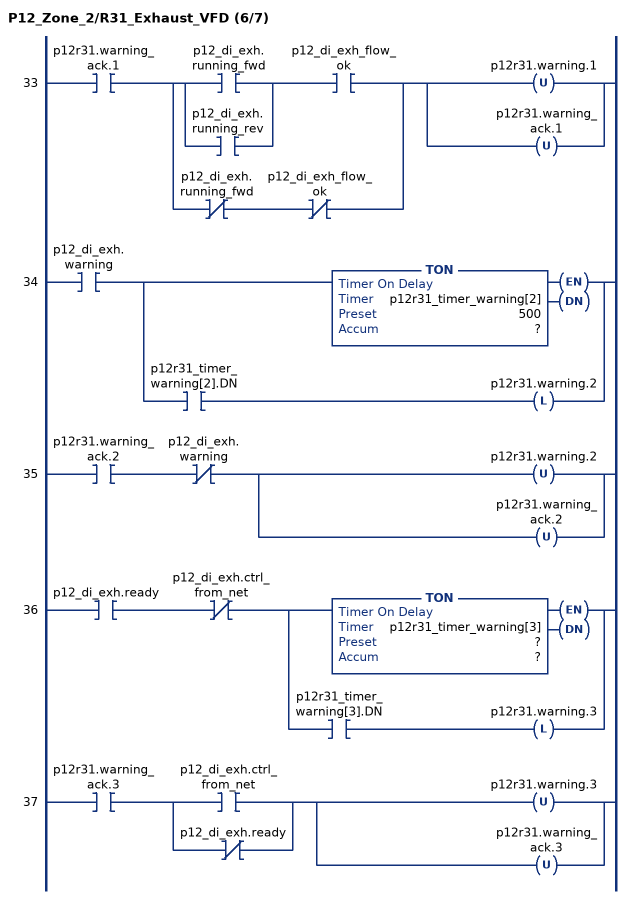
   33: XIC(p12r31.warning_ack.1)[[XIC(p12_di_exh.running_fwd) ,XIC(p12_di_exh.running_rev) ] XIC(p12_di_exh_flow_ok) ,XIO(p12_di_exh.running_fwd) XIO(p12_di_exh_flow_ok) ][OTU(p12r31.warning.1) ,OTU(p12r31.warning_ack.1) ];
   34: XIC(p12_di_exh.warning)[TON(p12r31_timer_warning[2],?,?) ,XIC(p12r31_timer_warning[2].DN) OTL(p12r31.warning.2) ];
   35: XIC(p12r31.warning_ack.2)XIO(p12_di_exh.warning)[OTU(p12r31.warning.2) ,OTU(p12r31.warning_ack.2) ];
   36: XIC(p12_di_exh.ready)XIO(p12_di_exh.ctrl_from_net)[TON(p12r31_timer_warning[3],?,?) ,XIC(p12r31_timer_warning[3].DN) OTL(p12r31.warning.3) ];
   37: XIC(p12r31.warning_ack.3)[XIC(p12_di_exh.ctrl_from_net) ,XIO(p12_di_exh.ready) ][OTU(p12r31.warning.3) ,OTU(p12r31.warning_ack.3) ];
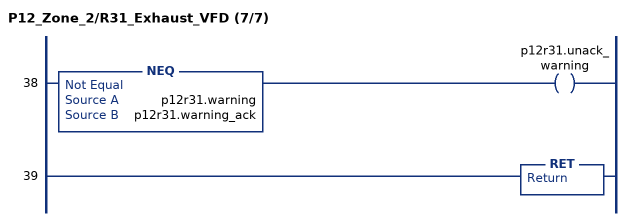
   38: NEQ(p12r31.warning,p12r31.warning_ack)OTE(p12r31.unack_warning);
   39: RET();
END_ROUTINE
